(* Logix 5000 project; controller cal1615 1756-L62 rev 20.11; software revision 20.05; part 44 of 81 *)
(* tags used below, declared in another part *)
   FAULT : BOOL;   // Fault AFI
   p01r09_pb_global_reset : BOOL;   // System Modes PB: Global Fault Reset
   p21_ai_splice_platen_temp : REAL;   // Splice Press Analog Input Platen Temperature
   p21_ao_splice_platen_temp_cv : REAL;   // Splice Press Analog Output Platen Temp Command Value
   p21_di_close_exit_clamp : BOOL;   // Splice Press Digital Input Close Exit Clamp
   p21_di_close_inlet_clamp : BOOL;   // Splice Press Digital Input Close Inlet Clamp
   p21_di_open_splice_platen : BOOL;   // Splice Press Digital Input Open Platen
   p21_di_platen_hi_temp_ok : BOOL;   // Splice Press Digital Input Platen High Temperature Ok
   p21_di_platen_not_closed : BOOL;   // Splice Press Digital Input Platen Not Closed
   p21_di_splice_2_hand_close : BOOL;   // Splice Press Digital Input Two Hand Switch Close Splicer
   p21_di_tc_bo : BOOL;   // Splice Press Digital Input Splice Platen Thermocouple Failure
   p21_dint_to_hmi : DINT[16];   // Splice Press
   p21_do_close_exit_clamp_sv : BOOL;   // Splice Press Digital Output Close Exit Clamp
   p21_do_close_inlet_clamp_sv : BOOL;   // Splice Press Digital Output Close Inlet Clamp
   p21_do_close_platen_sv : BOOL;   // Splice Press Digital Output Close Splicer Press
   p21_do_enable_platen_heater : BOOL;   // Splice Press Digital Output Enable Platen Heater
   p21_real_to_hmi : REAL[112];   // Splice Press Real to HMI
   p21_splice_press_temp_out : SYS_SCP;   // Splice Press Analog Ouputs Platen Heater
   p21_splice_temp_in_max : REAL;
   p21_splice_temp_in_min : REAL;
   p21_splice_temp_out_max : REAL;
   p21_splice_temp_out_min : REAL;
   P21r01 : routine;
   p21r03 : routine;   // Splice Press Inputs
   p21r03_timer_fault : TIMER[4];   // Splice Press Input Fault Dwell Timer
   p21r03_timer_warning : TIMER[4];   // Splice Press Input Warning Dwell Timer
   p21r04 : routine;   // Splice Press Outputs
   p21r04_timer_fault : TIMER[4];   // Splice Press Outputs Fault Delay
   p21r04_timer_warning : TIMER[4];   // Splice Press Outputs Warning Delay
   p21r05 : routine;   // Splice Press Dint to HMI
   p21r05_timer_fault : TIMER[4];   // Splice Press Dint to HMI Fault Delay
   p21r05_timer_warning : TIMER[4];   // Splice Press Dint to HMI Warning Delay
   p21r06 : routine;   // Splice Press Real to HMI
   p21r06_timer_fault : TIMER[4];   // Splice Press Real to HMI Fault Delay
   p21r06_timer_warning : TIMER[4];   // Splice Press Real to HMI Warning Delay
   p21r10_remaining_cure_time_sec : REAL;   // Splice Press Sequence Remaining Cure Timer [Sec]
   p21r10_status : DINT;   // Splice Press Sequence Status
   p21r16_pid_temp_cv : REAL;   // Splice Press Temperature Control PID Control Variable
   p21r16_request_heat : BOOL;   // Splice Press Temperature Control Request Heat
(* P21_Splice_Press, continued *)

ROUTINE R03_Input   (* ladder *)
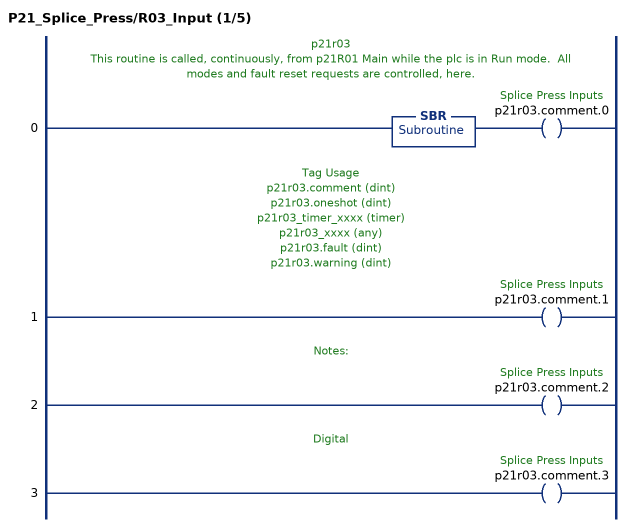
   // p21r03
   // This routine is called, continuously, from p21R01 Main while the plc is in Run mode.  All modes and fault reset requests are controlled, here.
   0: SBR()OTE(p21r03.comment.0);
   // Tag Usage
   // p21r03.comment (dint)
   // p21r03.oneshot (dint)
   // p21r03_timer_xxxx (timer)
   // p21r03_xxxx (any)
   // p21r03.fault (dint)
   // p21r03.warning (dint)
   1: OTE(p21r03.comment.1);
   // Notes:
   2: OTE(p21r03.comment.2);
   // Digital
   3: OTE(p21r03.comment.3);
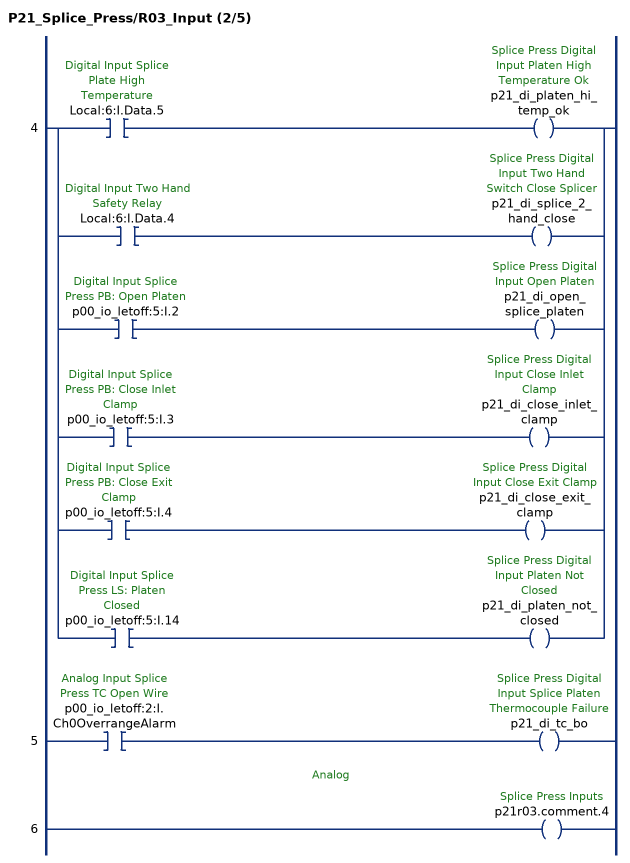
   4: [XIC(Local:6:I.Data.5) OTE(p21_di_platen_hi_temp_ok) ,XIC(Local:6:I.Data.4) OTE(p21_di_splice_2_hand_close) ,XIC(p00_io_letoff:5:I.2) OTE(p21_di_open_splice_platen) ,XIC(p00_io_letoff:5:I.3) OTE(p21_di_close_inlet_clamp) ,XIC(p00_io_letoff:5:I.4) OTE(p21_di_close_exit_clamp) ,XIC(p00_io_letoff:5:I.14) OTE(p21_di_platen_not_closed) ];
   5: XIC(p00_io_letoff:2:I.Ch0OverrangeAlarm)OTE(p21_di_tc_bo);
   // Analog
   6: OTE(p21r03.comment.4);
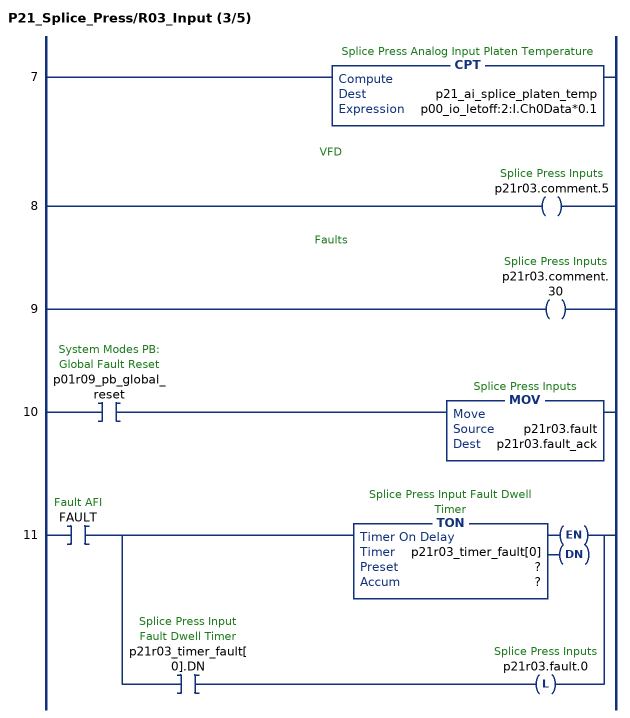
   7: CPT(p21_ai_splice_platen_temp,p00_io_letoff:2:I.Ch0Data*0.1);
   // VFD
   8: OTE(p21r03.comment.5);
   // Faults
   9: OTE(p21r03.comment.30);
   10: XIC(p01r09_pb_global_reset)MOV(p21r03.fault,p21r03.fault_ack);
   11: XIC(FAULT)[TON(p21r03_timer_fault[0],?,?) ,XIC(p21r03_timer_fault[0].DN) OTL(p21r03.fault.0) ];
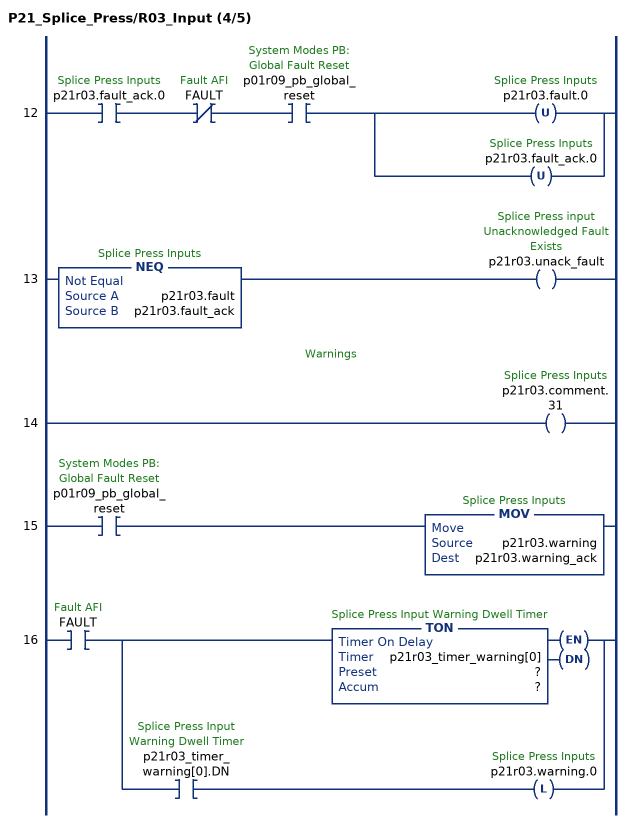
   12: XIC(p21r03.fault_ack.0)XIO(FAULT)XIC(p01r09_pb_global_reset)[OTU(p21r03.fault.0) ,OTU(p21r03.fault_ack.0) ];
   13: NEQ(p21r03.fault,p21r03.fault_ack)OTE(p21r03.unack_fault);
   // Warnings
   14: OTE(p21r03.comment.31);
   15: XIC(p01r09_pb_global_reset)MOV(p21r03.warning,p21r03.warning_ack);
   16: XIC(FAULT)[TON(p21r03_timer_warning[0],?,?) ,XIC(p21r03_timer_warning[0].DN) OTL(p21r03.warning.0) ];
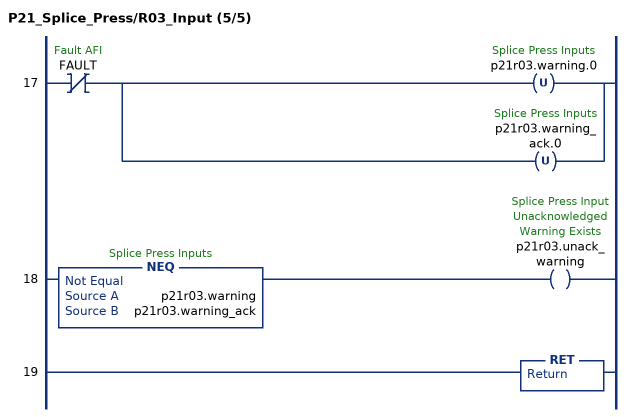
   17: XIO(FAULT)[OTU(p21r03.warning.0) ,OTU(p21r03.warning_ack.0) ];
   18: NEQ(p21r03.warning,p21r03.warning_ack)OTE(p21r03.unack_warning);
   19: RET();
END_ROUTINE

ROUTINE R04_Output   (* ladder *)
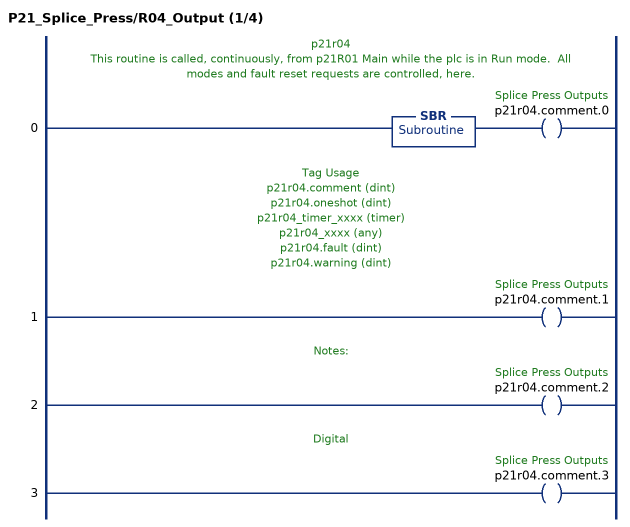
   // p21r04
   // This routine is called, continuously, from p21R01 Main while the plc is in Run mode.  All modes and fault reset requests are controlled, here.
   0: SBR()OTE(p21r04.comment.0);
   // Tag Usage
   // p21r04.comment (dint)
   // p21r04.oneshot (dint)
   // p21r04_timer_xxxx (timer)
   // p21r04_xxxx (any)
   // p21r04.fault (dint)
   // p21r04.warning (dint)
   1: OTE(p21r04.comment.1);
   // Notes:
   2: OTE(p21r04.comment.2);
   // Digital
   3: OTE(p21r04.comment.3);
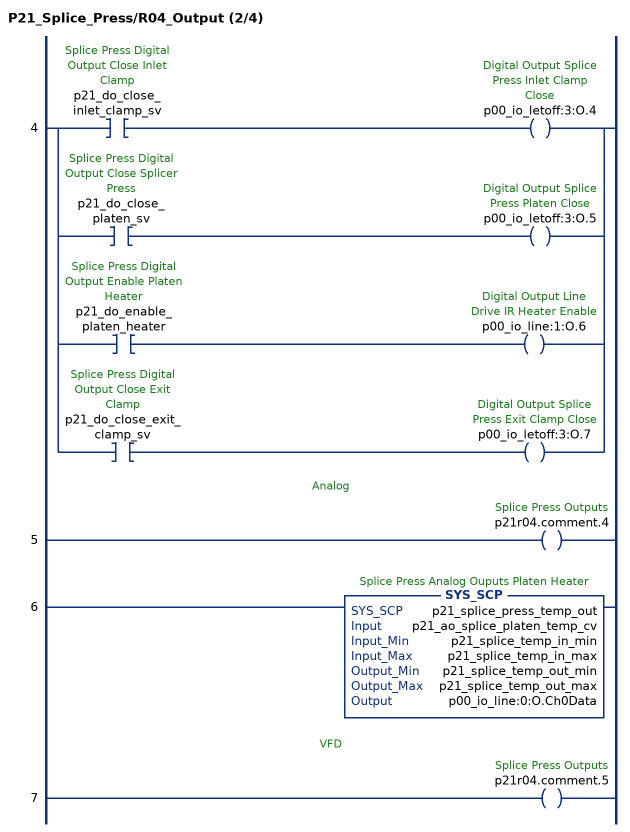
   4: [XIC(p21_do_close_inlet_clamp_sv) OTE(p00_io_letoff:3:O.4) ,XIC(p21_do_close_platen_sv) OTE(p00_io_letoff:3:O.5) ,XIC(p21_do_enable_platen_heater) OTE(p00_io_line:1:O.6) ,XIC(p21_do_close_exit_clamp_sv) OTE(p00_io_letoff:3:O.7) ];
   // Analog
   5: OTE(p21r04.comment.4);
   6: SYS_SCP(p21_splice_press_temp_out,p21_ao_splice_platen_temp_cv,p21_splice_temp_in_min,p21_splice_temp_in_max,p21_splice_temp_out_min,p21_splice_temp_out_max,p00_io_line:0:O.Ch0Data);
   // VFD
   7: OTE(p21r04.comment.5);
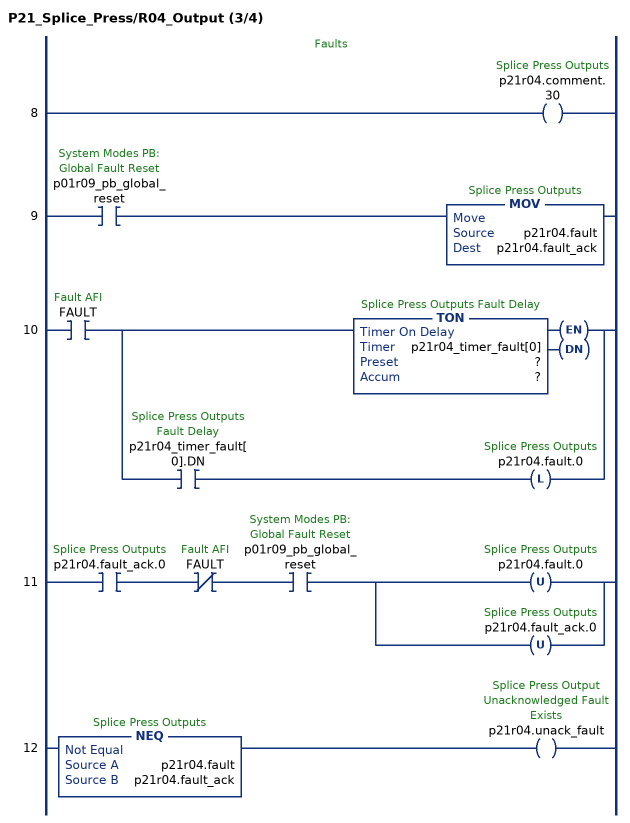
   // Faults
   8: OTE(p21r04.comment.30);
   9: XIC(p01r09_pb_global_reset)MOV(p21r04.fault,p21r04.fault_ack);
   10: XIC(FAULT)[TON(p21r04_timer_fault[0],?,?) ,XIC(p21r04_timer_fault[0].DN) OTL(p21r04.fault.0) ];
   11: XIC(p21r04.fault_ack.0)XIO(FAULT)XIC(p01r09_pb_global_reset)[OTU(p21r04.fault.0) ,OTU(p21r04.fault_ack.0) ];
   12: NEQ(p21r04.fault,p21r04.fault_ack)OTE(p21r04.unack_fault);
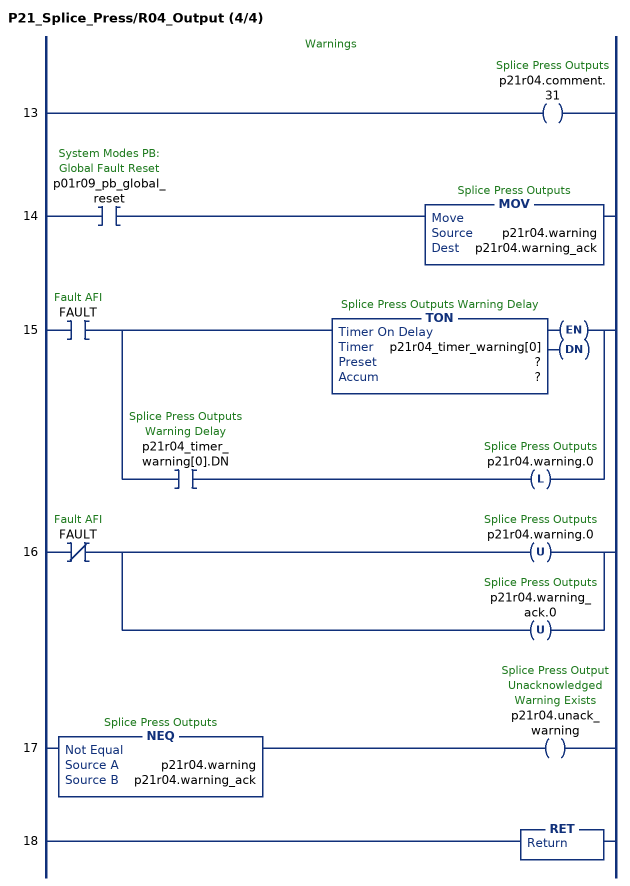
   // Warnings
   13: OTE(p21r04.comment.31);
   14: XIC(p01r09_pb_global_reset)MOV(p21r04.warning,p21r04.warning_ack);
   15: XIC(FAULT)[TON(p21r04_timer_warning[0],?,?) ,XIC(p21r04_timer_warning[0].DN) OTL(p21r04.warning.0) ];
   16: XIO(FAULT)[OTU(p21r04.warning.0) ,OTU(p21r04.warning_ack.0) ];
   17: NEQ(p21r04.warning,p21r04.warning_ack)OTE(p21r04.unack_warning);
   18: RET();
END_ROUTINE

ROUTINE R05_Dint_to_HMI   (* ladder *)
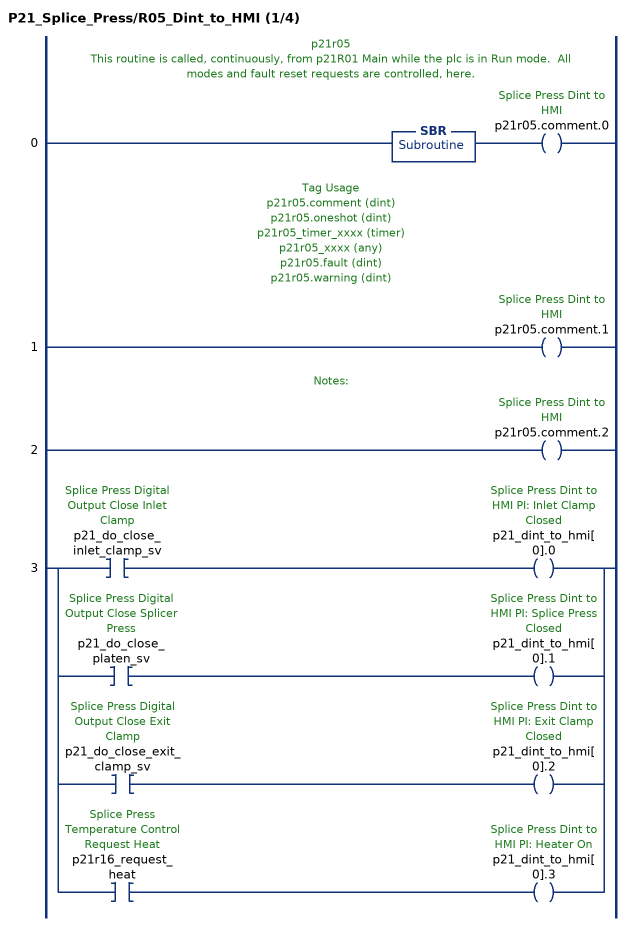
   // p21r05
   // This routine is called, continuously, from p21R01 Main while the plc is in Run mode.  All modes and fault reset requests are controlled, here.
   0: SBR()OTE(p21r05.comment.0);
   // Tag Usage
   // p21r05.comment (dint)
   // p21r05.oneshot (dint)
   // p21r05_timer_xxxx (timer)
   // p21r05_xxxx (any)
   // p21r05.fault (dint)
   // p21r05.warning (dint)
   1: OTE(p21r05.comment.1);
   // Notes:
   2: OTE(p21r05.comment.2);
   3: [XIC(p21_do_close_inlet_clamp_sv) OTE(p21_dint_to_hmi[0].0) ,XIC(p21_do_close_platen_sv) OTE(p21_dint_to_hmi[0].1) ,XIC(p21_do_close_exit_clamp_sv) OTE(p21_dint_to_hmi[0].2) ,XIC(p21r16_request_heat) OTE(p21_dint_to_hmi[0].3) ];
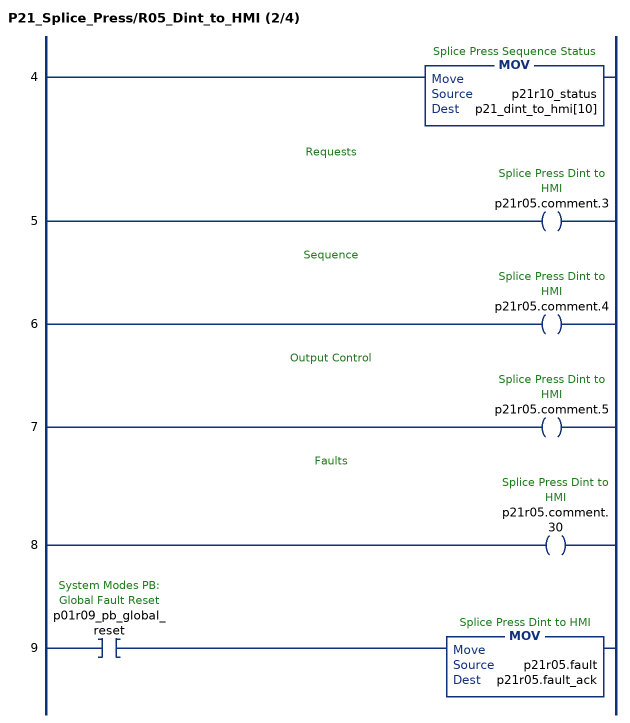
   4: MOV(p21r10_status,p21_dint_to_hmi[10]);
   // Requests
   5: OTE(p21r05.comment.3);
   // Sequence
   6: OTE(p21r05.comment.4);
   // Output Control
   7: OTE(p21r05.comment.5);
   // Faults
   8: OTE(p21r05.comment.30);
   9: XIC(p01r09_pb_global_reset)MOV(p21r05.fault,p21r05.fault_ack);
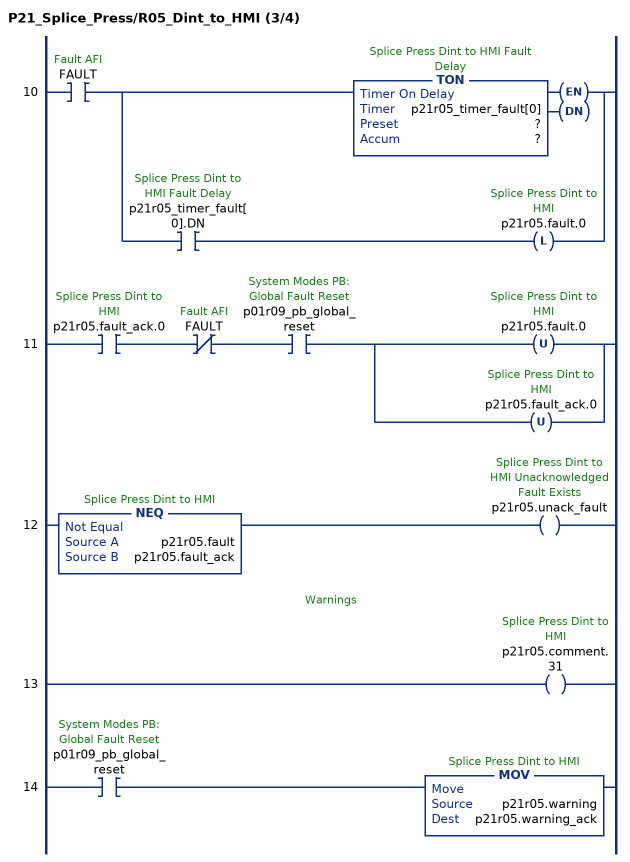
   10: XIC(FAULT)[TON(p21r05_timer_fault[0],?,?) ,XIC(p21r05_timer_fault[0].DN) OTL(p21r05.fault.0) ];
   11: XIC(p21r05.fault_ack.0)XIO(FAULT)XIC(p01r09_pb_global_reset)[OTU(p21r05.fault.0) ,OTU(p21r05.fault_ack.0) ];
   12: NEQ(p21r05.fault,p21r05.fault_ack)OTE(p21r05.unack_fault);
   // Warnings
   13: OTE(p21r05.comment.31);
   14: XIC(p01r09_pb_global_reset)MOV(p21r05.warning,p21r05.warning_ack);
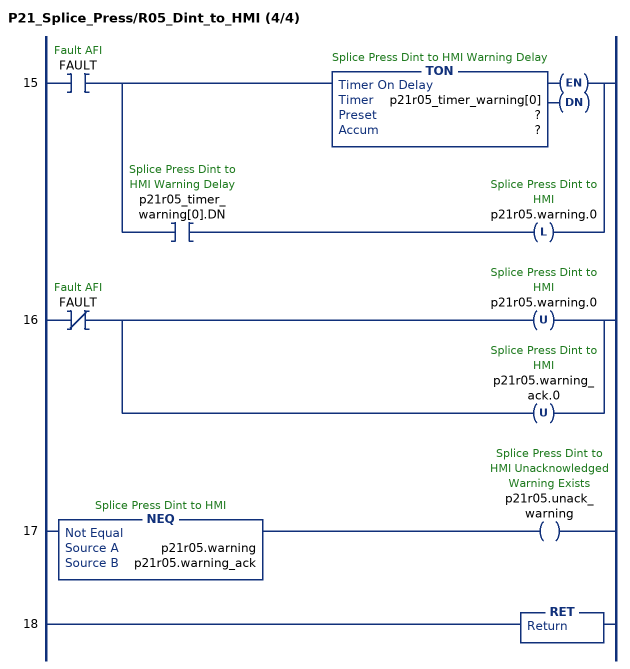
   15: XIC(FAULT)[TON(p21r05_timer_warning[0],?,?) ,XIC(p21r05_timer_warning[0].DN) OTL(p21r05.warning.0) ];
   16: XIO(FAULT)[OTU(p21r05.warning.0) ,OTU(p21r05.warning_ack.0) ];
   17: NEQ(p21r05.warning,p21r05.warning_ack)OTE(p21r05.unack_warning);
   18: RET();
END_ROUTINE

ROUTINE R06_Real_to_HMI   (* ladder *)
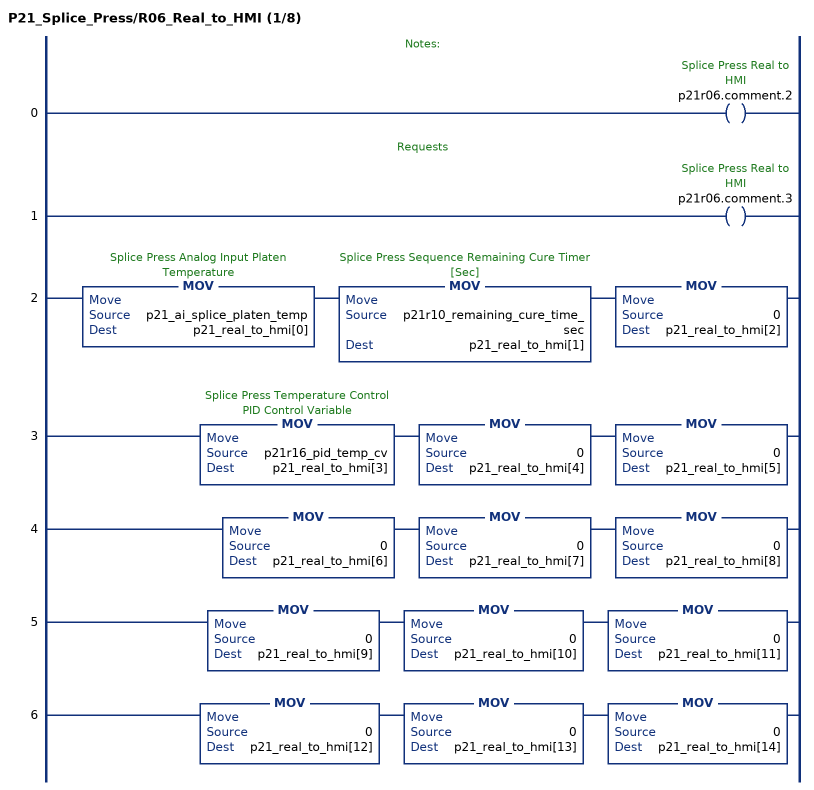
   // Notes:
   0: OTE(p21r06.comment.2);
   // Requests
   1: OTE(p21r06.comment.3);
   2: MOV(p21_ai_splice_platen_temp,p21_real_to_hmi[0])MOV(p21r10_remaining_cure_time_sec,p21_real_to_hmi[1])MOV(0,p21_real_to_hmi[2]);
   3: MOV(p21r16_pid_temp_cv,p21_real_to_hmi[3])MOV(0,p21_real_to_hmi[4])MOV(0,p21_real_to_hmi[5]);
   4: MOV(0,p21_real_to_hmi[6])MOV(0,p21_real_to_hmi[7])MOV(0,p21_real_to_hmi[8]);
   5: MOV(0,p21_real_to_hmi[9])MOV(0,p21_real_to_hmi[10])MOV(0,p21_real_to_hmi[11]);
   6: MOV(0,p21_real_to_hmi[12])MOV(0,p21_real_to_hmi[13])MOV(0,p21_real_to_hmi[14]);
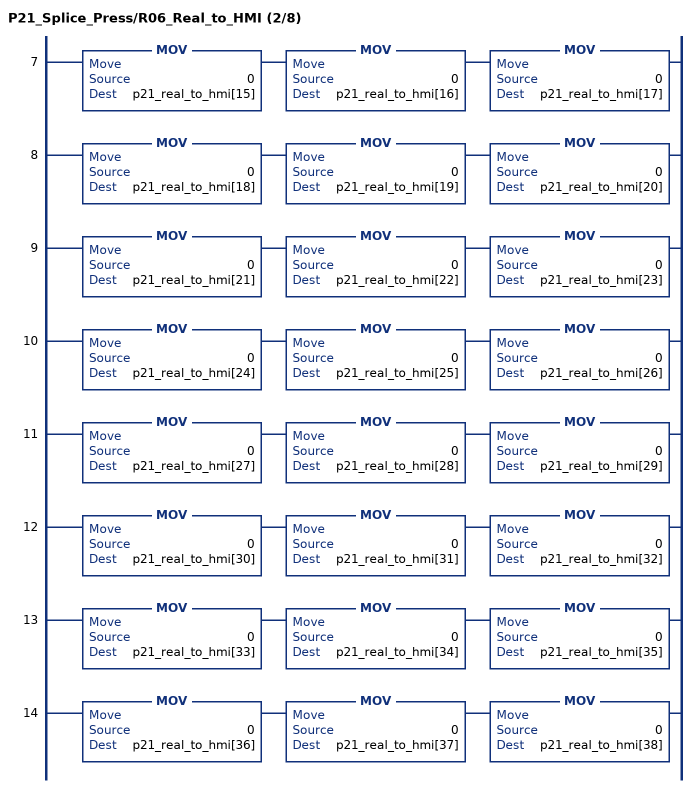
   7: MOV(0,p21_real_to_hmi[15])MOV(0,p21_real_to_hmi[16])MOV(0,p21_real_to_hmi[17]);
   8: MOV(0,p21_real_to_hmi[18])MOV(0,p21_real_to_hmi[19])MOV(0,p21_real_to_hmi[20]);
   9: MOV(0,p21_real_to_hmi[21])MOV(0,p21_real_to_hmi[22])MOV(0,p21_real_to_hmi[23]);
   10: MOV(0,p21_real_to_hmi[24])MOV(0,p21_real_to_hmi[25])MOV(0,p21_real_to_hmi[26]);
   11: MOV(0,p21_real_to_hmi[27])MOV(0,p21_real_to_hmi[28])MOV(0,p21_real_to_hmi[29]);
   12: MOV(0,p21_real_to_hmi[30])MOV(0,p21_real_to_hmi[31])MOV(0,p21_real_to_hmi[32]);
   13: MOV(0,p21_real_to_hmi[33])MOV(0,p21_real_to_hmi[34])MOV(0,p21_real_to_hmi[35]);
   14: MOV(0,p21_real_to_hmi[36])MOV(0,p21_real_to_hmi[37])MOV(0,p21_real_to_hmi[38]);
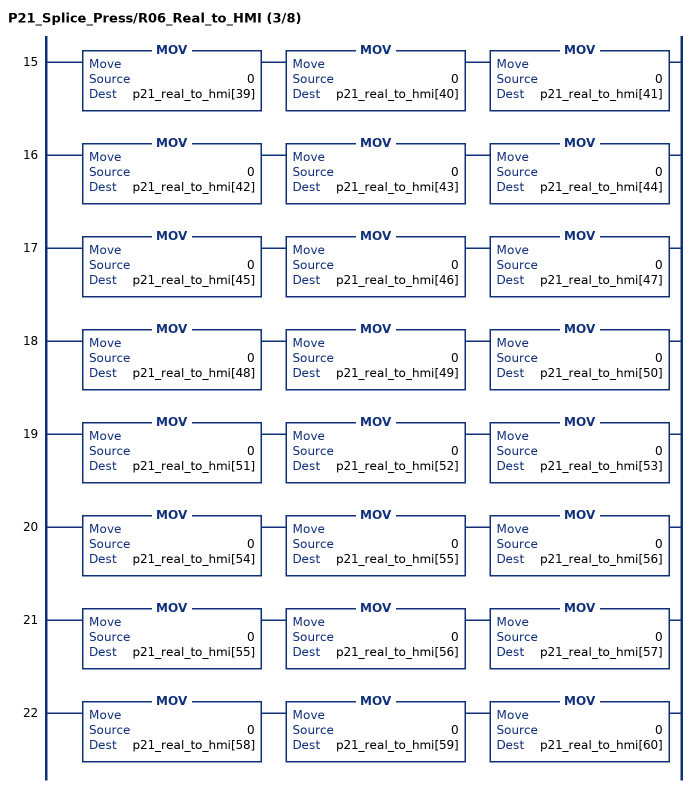
   15: MOV(0,p21_real_to_hmi[39])MOV(0,p21_real_to_hmi[40])MOV(0,p21_real_to_hmi[41]);
   16: MOV(0,p21_real_to_hmi[42])MOV(0,p21_real_to_hmi[43])MOV(0,p21_real_to_hmi[44]);
   17: MOV(0,p21_real_to_hmi[45])MOV(0,p21_real_to_hmi[46])MOV(0,p21_real_to_hmi[47]);
   18: MOV(0,p21_real_to_hmi[48])MOV(0,p21_real_to_hmi[49])MOV(0,p21_real_to_hmi[50]);
   19: MOV(0,p21_real_to_hmi[51])MOV(0,p21_real_to_hmi[52])MOV(0,p21_real_to_hmi[53]);
   20: MOV(0,p21_real_to_hmi[54])MOV(0,p21_real_to_hmi[55])MOV(0,p21_real_to_hmi[56]);
   21: MOV(0,p21_real_to_hmi[55])MOV(0,p21_real_to_hmi[56])MOV(0,p21_real_to_hmi[57]);
   22: MOV(0,p21_real_to_hmi[58])MOV(0,p21_real_to_hmi[59])MOV(0,p21_real_to_hmi[60]);
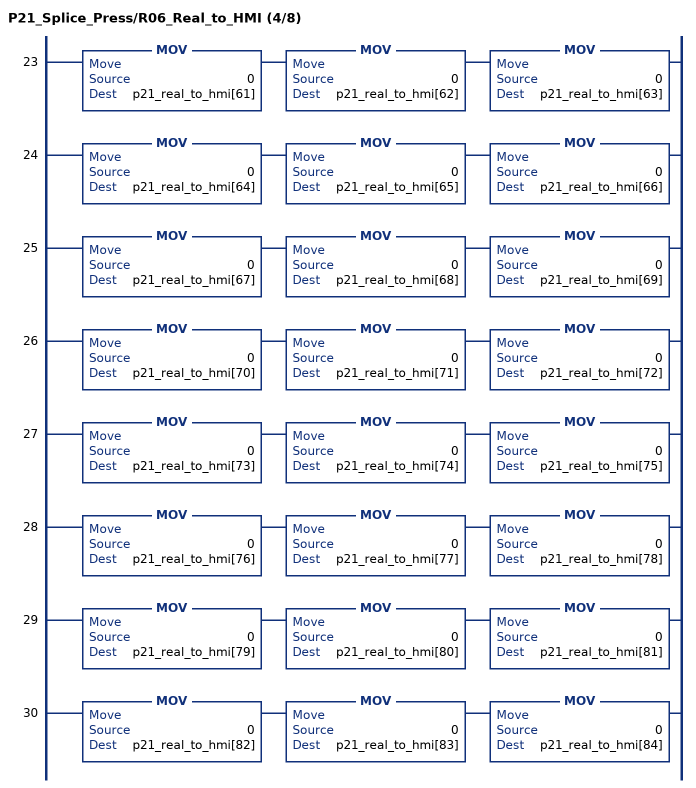
   23: MOV(0,p21_real_to_hmi[61])MOV(0,p21_real_to_hmi[62])MOV(0,p21_real_to_hmi[63]);
   24: MOV(0,p21_real_to_hmi[64])MOV(0,p21_real_to_hmi[65])MOV(0,p21_real_to_hmi[66]);
   25: MOV(0,p21_real_to_hmi[67])MOV(0,p21_real_to_hmi[68])MOV(0,p21_real_to_hmi[69]);
   26: MOV(0,p21_real_to_hmi[70])MOV(0,p21_real_to_hmi[71])MOV(0,p21_real_to_hmi[72]);
   27: MOV(0,p21_real_to_hmi[73])MOV(0,p21_real_to_hmi[74])MOV(0,p21_real_to_hmi[75]);
   28: MOV(0,p21_real_to_hmi[76])MOV(0,p21_real_to_hmi[77])MOV(0,p21_real_to_hmi[78]);
   29: MOV(0,p21_real_to_hmi[79])MOV(0,p21_real_to_hmi[80])MOV(0,p21_real_to_hmi[81]);
   30: MOV(0,p21_real_to_hmi[82])MOV(0,p21_real_to_hmi[83])MOV(0,p21_real_to_hmi[84]);
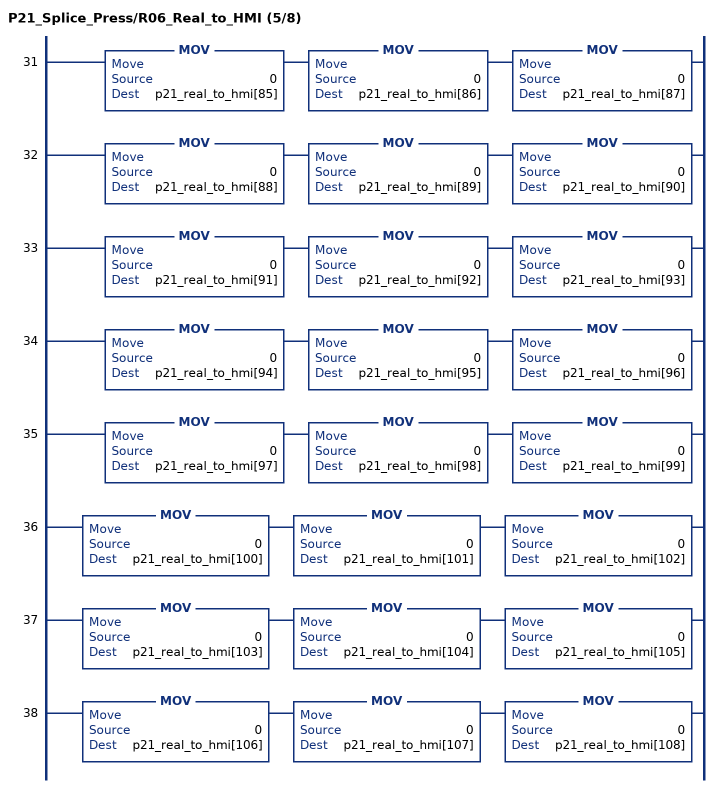
   31: MOV(0,p21_real_to_hmi[85])MOV(0,p21_real_to_hmi[86])MOV(0,p21_real_to_hmi[87]);
   32: MOV(0,p21_real_to_hmi[88])MOV(0,p21_real_to_hmi[89])MOV(0,p21_real_to_hmi[90]);
   33: MOV(0,p21_real_to_hmi[91])MOV(0,p21_real_to_hmi[92])MOV(0,p21_real_to_hmi[93]);
   34: MOV(0,p21_real_to_hmi[94])MOV(0,p21_real_to_hmi[95])MOV(0,p21_real_to_hmi[96]);
   35: MOV(0,p21_real_to_hmi[97])MOV(0,p21_real_to_hmi[98])MOV(0,p21_real_to_hmi[99]);
   36: MOV(0,p21_real_to_hmi[100])MOV(0,p21_real_to_hmi[101])MOV(0,p21_real_to_hmi[102]);
   37: MOV(0,p21_real_to_hmi[103])MOV(0,p21_real_to_hmi[104])MOV(0,p21_real_to_hmi[105]);
   38: MOV(0,p21_real_to_hmi[106])MOV(0,p21_real_to_hmi[107])MOV(0,p21_real_to_hmi[108]);
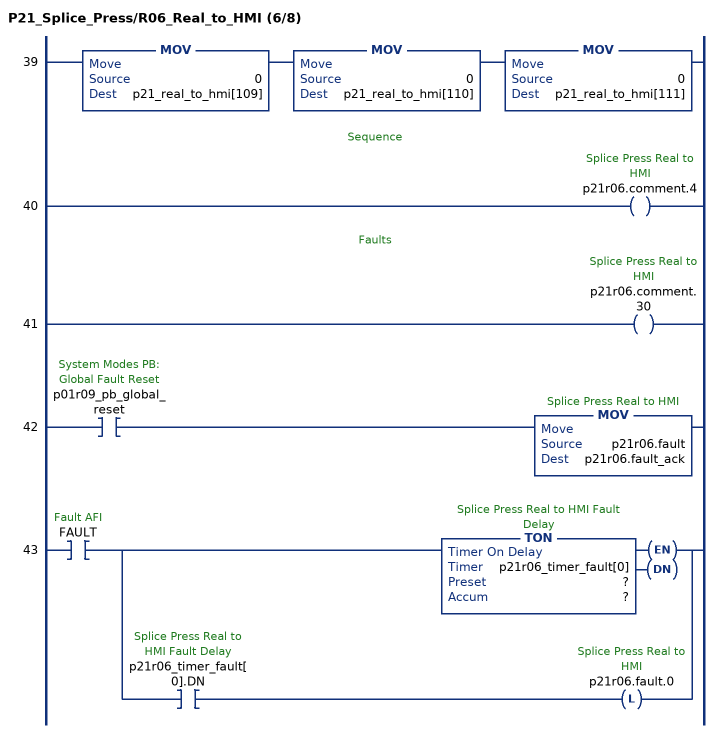
   39: MOV(0,p21_real_to_hmi[109])MOV(0,p21_real_to_hmi[110])MOV(0,p21_real_to_hmi[111]);
   // Sequence
   40: OTE(p21r06.comment.4);
   // Faults
   41: OTE(p21r06.comment.30);
   42: XIC(p01r09_pb_global_reset)MOV(p21r06.fault,p21r06.fault_ack);
   43: XIC(FAULT)[TON(p21r06_timer_fault[0],?,?) ,XIC(p21r06_timer_fault[0].DN) OTL(p21r06.fault.0) ];
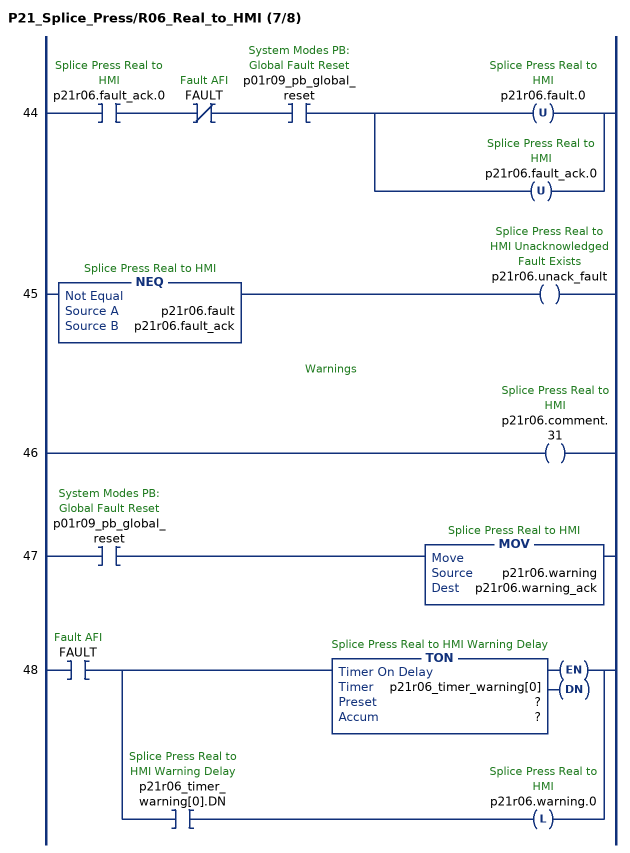
   44: XIC(p21r06.fault_ack.0)XIO(FAULT)XIC(p01r09_pb_global_reset)[OTU(p21r06.fault.0) ,OTU(p21r06.fault_ack.0) ];
   45: NEQ(p21r06.fault,p21r06.fault_ack)OTE(p21r06.unack_fault);
   // Warnings
   46: OTE(p21r06.comment.31);
   47: XIC(p01r09_pb_global_reset)MOV(p21r06.warning,p21r06.warning_ack);
   48: XIC(FAULT)[TON(p21r06_timer_warning[0],?,?) ,XIC(p21r06_timer_warning[0].DN) OTL(p21r06.warning.0) ];
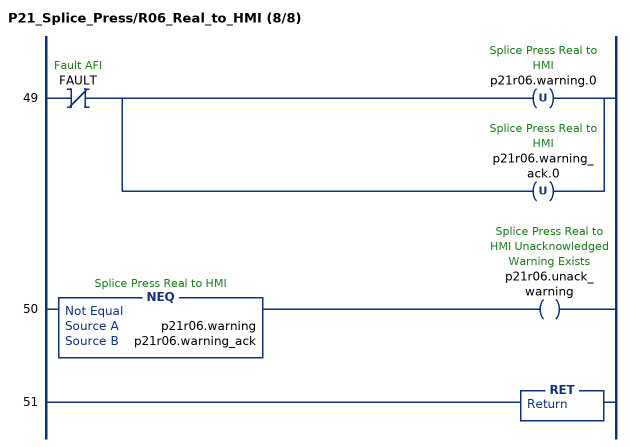
   49: XIO(FAULT)[OTU(p21r06.warning.0) ,OTU(p21r06.warning_ack.0) ];
   50: NEQ(p21r06.warning,p21r06.warning_ack)OTE(p21r06.unack_warning);
   51: RET();
END_ROUTINE
